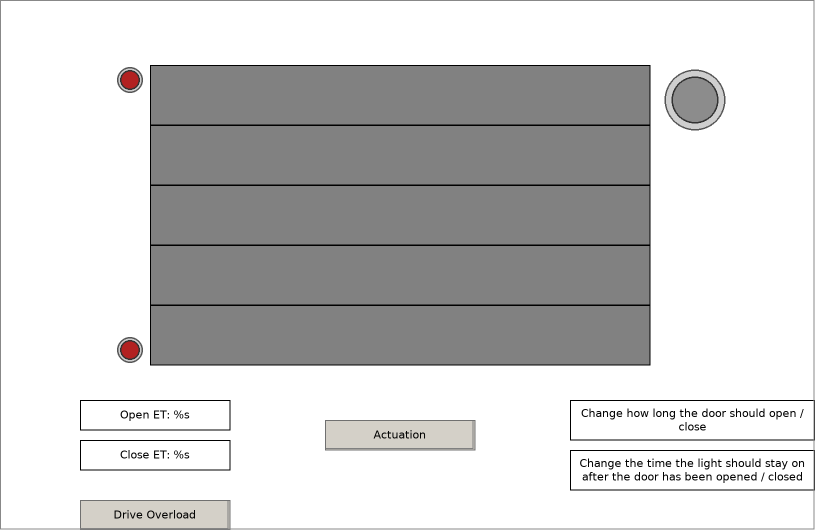
VISUALIZATION Visualization  // 815x530
    Button (325,420 150x30), "Actuation"
        tap MAIN.bButtonPress
    Lamp1 (660,65 70x70), variable: MAIN.fbActuation.bDoorLight, style: Lamp-Lamp1-Gray
    Rectangle (80,400 150x30), "Open ET: %s", text variable: MAIN.fbActuation.fbOpeningTimer.ET
    Rectangle (80,440 150x30), "Close ET: %s", text variable: MAIN.fbActuation.fbClosingTimer.ET
    Rectangle (150,65 500x300)
    Rectangle (150,65 500x60), invisible if: MAIN.fbActuation.Rect5
    Rectangle (150,125 500x60), invisible if: MAIN.fbActuation.Rect4
    Rectangle (150,185 500x60), invisible if: MAIN.fbActuation.Rect3
    Rectangle (150,245 500x60), invisible if: MAIN.fbActuation.Rect2
    Rectangle (150,305 500x60), invisible if: MAIN.fbActuation.Rect1
    Lamp1 (115,65 30x30), variable: MAIN.fbActuation.bDoorOpen, style: Lamp-Lamp1-Red
    Lamp1 (115,335 30x30), variable: MAIN.fbActuation.bDoorClosed, style: Lamp-Lamp1-Red
    Button (80,500 150x30), "Drive Overload"
        tap MAIN.fbActuation.bDriveOverload
    Rectangle (570,450 245x40), "Change the time the light should stay on after the door has been opened / closed"
        OnMouseClick: write MAIN.fbActuation.LIGHT_DELAY via Default
    Rectangle (570,400 245x40), "Change how long the door should open / close"
        OnMouseClick: write MAIN.fbActuation.TIMER_PRESET via Default
END_VISUALIZATION

(* stored: Version 1.1.0.1, ProductVersion 3.1.4024.12
   Visu Visualization: Id {3a8afb4d-9d8b-4460-b3cc-3026ddc30c29} *)
